ABB RobotStudio station: basith material handling_2.rsstn

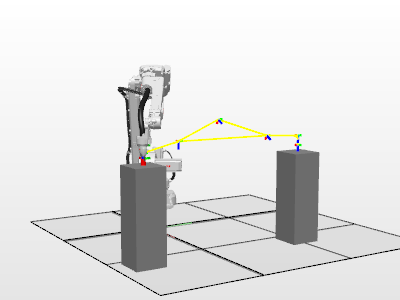
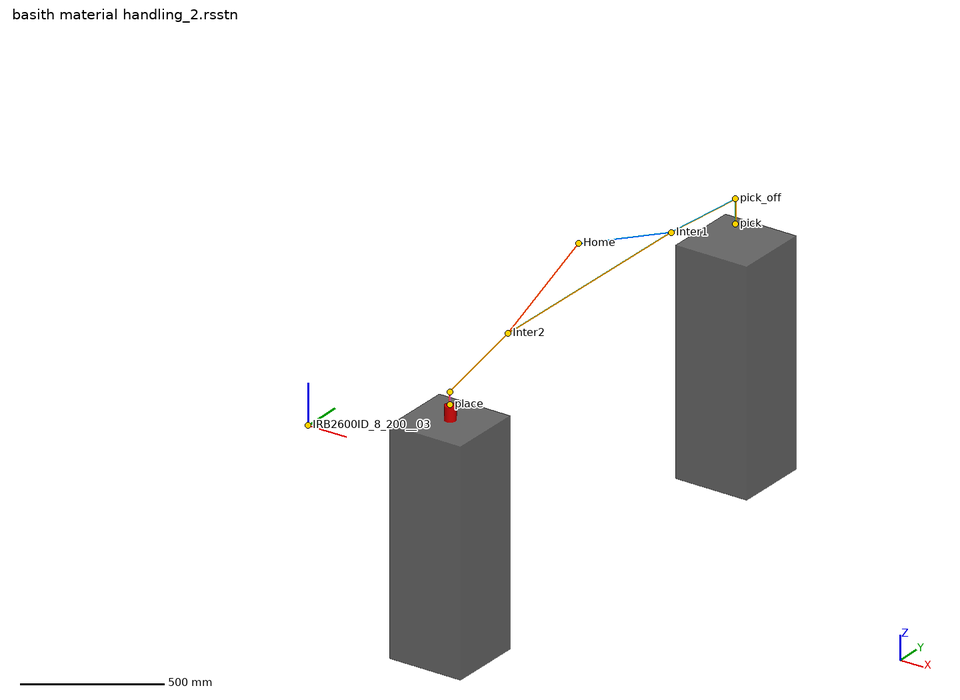
[picture v1: parts stored in the station drawn from their meshes, with robot base, taught points and paths (robot models come from the ABB library and are not in the file)]
Station eshwaran material handling_1 (saved by RobotStudio 22.3.10141.1)
Controller Controller6, task T_ROB1: task frame (RAPID world) sits at (96.74, 0, 279.25) mm in the station
Controller Controller6
  mechanical unit ROB_1: IRB2600ID_8_200__03, 6 joints, base frame (0, 0, 0) mm
Layout (positions relative to the parent item):
  - IRB2600ID_8_200__03 [mechanism, from %ABB.RobotStudio.Models.IRB2600ID%\IRB2600ID_8_200_G_03.rslib] at (96.74, 0, 279.25) mm; joint values [-0.5816, 0.3097, 0.1782, 0.0055, 1.0755, -0.5842] (rad or m)
  - SmartComponent_1 [smart component]
      signals: DI attach
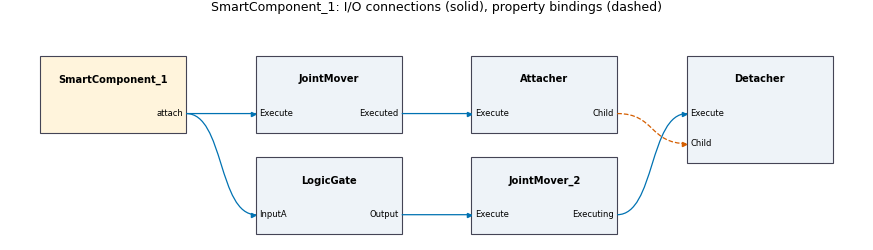
      connections:
        SmartComponent_1.attach -> JointMover.Execute
        JointMover.Executed -> Attacher.Execute
        SmartComponent_1.attach -> LogicGate.InputA
        LogicGate.Output -> JointMover_2.Execute
        JointMover_2.Executing -> Detacher.Execute
        Attacher.Child => Detacher.Child
    - Smart_Gripper_Servo_Fingers [mechanism, from Tools\ABB_Smart_Gripper_Servo_Fingers.rslib] at (1204.14, -726.94, 1074.2) mm, rotated rx 180 ry 0.51 rz -180 deg; joint values [0.025] (rad or m)
    - Attacher [smart component, from Components\Attacher.rslib]
        properties: Parent=Smart_Gripper_Servo_Fingers; Flange=0; Child=Part_4; Mount=false; Offset=[0 0 0]; Orientation=[0 0 0]
    - Detacher [smart component, from Components\Detacher.rslib]
        properties: Child=Part_4; KeepPosition=true
    - JointMover [smart component, from Components\JointMover.rslib]
        properties: Mechanism=Smart_Gripper_Servo_Fingers; Relative=false; Duration=0; J1=0.023
    - JointMover_2 [smart component, from Components\JointMover.rslib]
        properties: Mechanism=Smart_Gripper_Servo_Fingers; Relative=false; Duration=0; J1=0.025
    - LogicGate [smart component, from Components\LogicGate.rslib]
        properties: Operator=NOT; Delay=0
  - Table 1 [part] at (1051.6, 857.35, 0) mm, size 300 x 300 x 900 mm
  - Table 1_3 [part] at (1055.16, -876.94, 0) mm, size 300 x 300 x 900 mm
  - Part_4 [part] at (1205.16, -724, 896.21) mm, size 45 x 44.7 x 60 mm
  - Part_5 [part] at (1205.16, -726.94, 900) mm, size 45 x 44.7 x 60 mm
Attachment: Smart_Gripper_Servo_Fingers is attached to IRB2600ID_8_200__03 / Link6
Station logic (signal -> signal, property => property):
  Controller6.Attach -> SmartComponent_1.attach
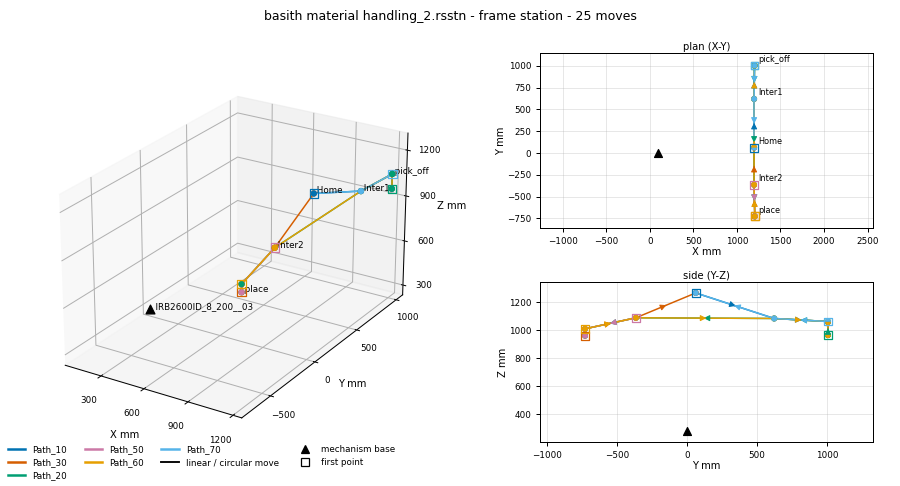
[picture p0: tool path of basith material handling_2.rsstn in frame station, 25 of 25 moves have a stored position in this frame; points joined in program order, loops and branches not executed]
Targets, tools, work objects and paths stored in the station, written as RAPID:
! task T_ROB1
MODULE CalibData
  PERS tooldata Servo:=[TRUE,[[0,0,114.2],[1,0,0,0]],[0.215,[8.7,12.3,49.2],[1,0,0,0],0.00021,0.00024,0.00009]];
ENDMODULE

! task T_ROB1
MODULE Module1
  CONST robtarget Home:=[[1100.818000968,61.948263808,985.403234621],[0.500000012,-0.00000005,0.866025397,0.000000009],[0,-1,0,0],[9E+09,9E+09,9E+09,9E+09,9E+09,9E+09]];
  CONST robtarget Inter1:=[[1100.818014371,620.944035019,803.451786818],[0.500000016,-0.000000039,0.866025394,0.000000037],[0,-1,1,0],[9E+09,9E+09,9E+09,9E+09,9E+09,9E+09]];
  CONST robtarget pick:=[[1104.861027808,1004.407035703,684.547469003],[0.004443238,-0.000000123,0.999990129,0.000000075],[0,-1,0,0],[9E+09,9E+09,9E+09,9E+09,9E+09,9E+09]];
  CONST robtarget pick_off:=[[1104.861007274,1004.407016755,781.60740596],[0.00444322,-0.000000105,0.999990129,0.000000058],[0,-1,0,0],[9E+09,9E+09,9E+09,9E+09,9E+09,9E+09]];
  CONST robtarget Inter2:=[[1100.252970882,-364.502312698,808.320329719],[0.004443315,-0.00000008,0.999990128,0.000000084],[-1,0,-1,0],[9E+09,9E+09,9E+09,9E+09,9E+09,9E+09]];
  CONST robtarget place:=[[1108.412009128,-726.941796168,680.753856958],[0.00444332,-0.000000109,0.999990128,0.000000081],[-1,0,-1,0],[9E+09,9E+09,9E+09,9E+09,9E+09,9E+09]];
  CONST robtarget placeoff:=[[1108.412003536,-726.941792416,729.622335546],[0.004443299,-0.000000118,0.999990128,0.000000095],[-1,0,-1,0],[9E+09,9E+09,9E+09,9E+09,9E+09,9E+09]];
  PROC Path_10()
    MoveL Home,v1000,z100,Servo\WObj:=wobj0;
    MoveL Inter1,v1000,z100,Servo\WObj:=wobj0;
    MoveL pick_off,v1000,z100,Servo\WObj:=wobj0;
    MoveL pick,v1000,z100,Servo\WObj:=wobj0;
    WaitTime 1;
    SetDO Attach,1;
    WaitTime 1;
  ENDPROC
  PROC Path_30()
    MoveL place,v1000,z100,Servo\WObj:=wobj0;
    MoveL placeoff,v1000,z100,Servo\WObj:=wobj0;
    MoveL Inter2,v1000,z100,Servo\WObj:=wobj0;
    MoveL Home,v1000,z100,Servo\WObj:=wobj0;
  ENDPROC
  PROC Path_20()
    MoveL pick,v1000,z100,Servo\WObj:=wobj0;
    MoveL pick_off,v1000,z100,Servo\WObj:=wobj0;
    MoveL Inter1,v1000,z100,Servo\WObj:=wobj0;
    MoveL Inter2,v1000,z100,Servo\WObj:=wobj0;
    MoveL placeoff,v1000,z100,Servo\WObj:=wobj0;
    MoveL place,v1000,z100,Servo\WObj:=wobj0;
    WaitTime 1;
    SetDO Attach,0;
    WaitTime 1;
  ENDPROC
  PROC Path_40()
    Path_10;
    Path_20;
    Path_50;
    Path_30;
    Path_60;
    Path_70;
  ENDPROC
  PROC Path_50()
    MoveL Inter2,v1000,z100,Servo\WObj:=wobj0;
    MoveL placeoff,v1000,z100,Servo\WObj:=wobj0;
    MoveL place,v1000,z100,Servo\WObj:=wobj0;
    SetDO Attach,1;
    WaitTime 1;
    WaitTime 1;
  ENDPROC
  PROC Path_60()
    MoveL placeoff,v1000,z100,Servo\WObj:=wobj0;
    MoveL Inter2,v1000,z100,Servo\WObj:=wobj0;
    MoveL Inter1,v1000,z100,Servo\WObj:=wobj0;
    MoveL pick_off,v1000,z100,Servo\WObj:=wobj0;
    MoveL pick,v1000,z100,Servo\WObj:=wobj0;
    WaitTime 1;
    SetDO Attach,0;
    WaitTime 1;
  ENDPROC
  PROC Path_70()
    MoveL pick_off,v1000,z100,Servo\WObj:=wobj0;
    MoveL Inter1,v1000,z100,Servo\WObj:=wobj0;
    MoveL Home,v1000,z100,Servo\WObj:=wobj0;
  ENDPROC
ENDMODULE

